// TIA Portal V17 export
// export: Created 2025-06-26T06:33:53.9939344Z, ExportSetting WithDefaults, DisplayName Totally Integrated Automation Portal, DisplayVersion V17 Update 8, DisplayName TIA Portal Openness, DisplayVersion V17 Update 8, DisplayName TIA Portal Version Control Interface, DisplayVersion V17, DisplayName STEP 7 Professional, DisplayVersion V17 Update 8, DisplayName STEP 7 Safety, DisplayVersion V17 Update 6, DisplayName WinCC Advanced, DisplayVersion V17 Update 8
DATA_BLOCK "CAN_Data_DB"   // DB3
{ S7_Optimized_Access := 'TRUE' }
VERSION : 0.1
// stored: AutoNumber true, DBAccessibleFromOPCUA true, IsOnlyStoredInLoadMemory false, IsRetainMemResEnabled false, IsWriteProtectedInAS false, MemoryReserve 100
   VAR
      InputData : Struct   // Receive
         CAN_ID_101h : Struct
            StartRequest : Bool;
            StopRequest : Bool;
            Clearance : Bool;
            PumaSystemReady : Bool;
            AlarmAcknowledge : Bool;
            ResetEmergencyStop : Bool;
            FastStopRequest : Bool;
            HydrolockProtection : Bool;
            ForceSuperheatSP : Bool;
            ForceHeatSinkOutSP : Bool;
            ForcePerformanceControlSP : Bool;
            ForceOilHeatingSP : Bool;
            ForceExpansionValveSP : Bool;
            ForcePinchSP : Bool;
            SpareByte2Bit6 : Bool;
            SpareByte2Bit7 : Bool;
            WatchdogFeedback : Word;
            I_326 : Bool;   // 0
            I_327 : Bool;   // 1
            I_330 : Bool;   // 2
            I_372 : Bool;   // 3
            I_373 : Bool;   // 4
            Spare55 : Bool;   // 5
            Spare56 : Bool;   // 6
            Spare57 : Bool;   // 7
            Spare60 : Bool;   // 0
            Spare61 : Bool;   // 1
            Spare62 : Bool;   // 2
            Spare63 : Bool;   // 3
            Spare64 : Bool;   // 4
            Spare65 : Bool;   // 5
            Spare66 : Bool;   // 6
            Spare67 : Bool;   // 7
            SpareByte7 : Byte;
            SpareByte8 : Byte;
         END_STRUCT;
         CAN_ID_102h : Struct
            SuperheatSP : Real;
            HeatSinkOutSP : Real;
         END_STRUCT;
         CAN_ID_103h : Struct
            PerformanceControlSP : Real;
            OilHeatingSP : Real;
         END_STRUCT;
         CAN_ID_104h : Struct
            ExpansionValveSP : Real;
            PinchSP : Real;
         END_STRUCT;
         CAN_ID_105h : Struct
            ThermalPowerOutput : Real;
            ThermalPowerInput : Real;
         END_STRUCT;
         CAN_ID_110h : Struct
            I_208 : Real;
            I_209 : Real;
         END_STRUCT;
         CAN_ID_111h : Struct
            I_210 : Real;
            I_211 : Real;
         END_STRUCT;
         CAN_ID_112h : Struct
            I_206 : Real;
            E_214 : Real;
         END_STRUCT;
         CAN_ID_113h : Struct
            I_302 : Real;
            E_213 : Real;
         END_STRUCT;
         CAN_ID_114h : Struct
            I_301 : Real;
            I_201 : Real;
         END_STRUCT;
         CAN_ID_115h : Struct
            I_202 : Real;
            I_307 : Real;
         END_STRUCT;
         CAN_ID_116h : Struct
            I_355 : Real;
            I_308 : Real;
         END_STRUCT;
         CAN_ID_117h : Struct
            I_300 : Real;
            I_301 : Real;
         END_STRUCT;
         CAN_ID_118h : Struct
            I_304 : Real;
            I_306 : Real;
         END_STRUCT;
         CAN_ID_119h : Struct
            I_320 : Real;
            I_321 : Real;
         END_STRUCT;
         CAN_ID_120h : Struct
            I_322 : Real;
            I_323 : Real;
         END_STRUCT;
         CAN_ID_121h : Struct
            I_324 : Real;
            I_328 : Real;
         END_STRUCT;
         CAN_ID_122h : Struct
            I_350 : Real;
            I_351 : Real;
         END_STRUCT;
         CAN_ID_123h : Struct
            I_354 : Real;
            I_356 : Real;
         END_STRUCT;
         CAN_ID_124h : Struct
            I_370 : Real;
            I_374 : Real;
         END_STRUCT;
         CAN_ID_125h : Struct
            E_301 : Real;
            E_330 : Real;
         END_STRUCT;
         CAN_ID_126h : Struct
            E_351 : Real;
            Spare : Real;
         END_STRUCT;
      END_STRUCT;
      OutputData { S7_SetPoint := 'True'} : "CAN-IDs_ToSend";   // Send
   END_VAR
BEGIN
   OutputData.IDs[5] := 16#0210;
   OutputData.IDs[6] := 16#0211;
   OutputData.IDs[7] := 16#0212;
   OutputData.IDs[8] := 16#0213;
   OutputData.IDs[9] := 16#0214;
   OutputData.IDs[10] := 16#0215;
   OutputData.IDs[11] := 16#0216;
   OutputData.IDs[12] := 16#0217;
   OutputData.IDs[13] := 16#0218;
   OutputData.IDs[14] := 16#0219;
   OutputData.IDs[15] := 16#0220;
   OutputData.IDs[16] := 16#0221;
   OutputData.IDs[17] := 16#0222;
   OutputData.IDs[18] := 16#0223;
   OutputData.IDs[19] := 16#0224;
   OutputData.IDs[20] := 16#0225;
   OutputData.IDs[21] := 16#0226;
   OutputData.IDs[22] := 16#0227;
   OutputData.IDs[23] := 16#0228;
   OutputData.IDs[24] := 16#0229;
   OutputData.IDs[25] := 16#0231;
   OutputData.IDs[26] := 16#0232;
   OutputData.IDs[27] := 16#0235;
   OutputData.IDs[28] := 16#0236;
   OutputData.IDs[29] := 16#0237;
   OutputData.IDs[30] := 16#0238;
   OutputData.IDs[31] := 16#0239;
   OutputData.IDs[32] := 16#0240;
   OutputData.IDs[33] := 16#0241;
   OutputData.IDs[34] := 16#0242;
   OutputData.IDs[35] := 16#0243;
   OutputData.IDs[36] := 16#0244;
   OutputData.IDs[37] := 16#0245;
   OutputData.IDs[38] := 16#0246;
   OutputData.IDs[39] := 16#0247;
   OutputData.IDs[40] := 16#0248;
   OutputData.IDs[41] := 16#0250;
   OutputData.IDs[42] := 16#0251;
   OutputData.IDs[43] := 16#0252;
   OutputData.IDs[44] := 16#0253;
   OutputData.IDs[45] := 16#0254;
   OutputData.IDs[46] := 16#0255;
   OutputData.IDs[47] := 16#0256;
   OutputData.IDs[48] := 16#0257;
   OutputData.IDs[49] := 16#0258;
   OutputData.IDs[50] := 16#0259;
   OutputData.IDs[51] := 16#0260;
   OutputData.IDs[52] := 16#0261;
   OutputData.IDs[53] := 16#0262;
   OutputData.IDs[54] := 16#0263;
   OutputData.IDs[55] := 16#0264;
   OutputData.IDs[56] := 16#0265;
   OutputData.IDs[57] := 16#0266;
   OutputData.IDs[58] := 16#0301;
   OutputData.IDs[59] := 16#0302;
   OutputData.IDs[60] := 16#0303;
   OutputData.IDs[61] := 16#0304;
   OutputData.IDs[62] := 16#0311;
   OutputData.IDs[63] := 16#0312;
   OutputData.IDs[64] := 16#0313;
   OutputData.IDs[65] := 16#0314;
   OutputData.IDs[66] := 16#0315;
   OutputData.IDs[67] := 16#0305;
   OutputData.IDs[68] := 16#0230;
END_DATA_BLOCK
